(* PLC project OOP_Curso, Beckhoff Automation GmbH TwinCAT PLC Control 3.5.13.21 *)
(* stored: creationDateTime 2023-06-14T13:02:06.5620853, modificationDateTime 2023-06-14T13:02:06.5620853 *)

(* global variable list GVL_Exc *)
{attribute 'qualified_only'}
VAR_GLOBAL CONSTANT
    cMaxExc            : UINT := 10;
END_VAR
VAR_GLOBAL
    nExcIndex          : UINT;
    aExceptionHistory  : ARRAY[0..cMaxExc] OF __SYSTEM.ExceptionCode;
END_VAR

(* global variable list GVL *)
{attribute 'qualified_only'}
VAR_GLOBAL
    bGlobalTestFlag : BOOL;
END_VAR

INTERFACE I_Base EXTENDS __SYSTEM.IQueryInterface
METHOD Base : BOOL
VAR_INPUT
END_VAR
END_METHOD
END_INTERFACE

INTERFACE I_Derived EXTENDS I_Base
METHOD Derived : BOOL
VAR_INPUT
END_VAR
END_METHOD
END_INTERFACE

FUNCTION_BLOCK FB_Variante IMPLEMENTS I_Derived
VAR_INPUT
END_VAR
VAR_OUTPUT
END_VAR
VAR
END_VAR

            
          

{warning 'add method implementation '}
METHOD Base : BOOL
                  
                
END_METHOD

{warning 'add method implementation '}
METHOD Derived : BOOL
                  
                
END_METHOD
END_FUNCTION_BLOCK

PROGRAM QUERYPOINTER
//__QUERYPOINTER
VAR
    iDerived   : I_Derived;
    fbVariante : FB_Variante;
    bResult    : BOOL;
    bTest      : BOOL;
    pFB        : POINTER TO FB_Variante;
END_VAR

            //__QUERYPOINTER
iDerived := fbVariante;
bResult  := __QUERYPOINTER(iDerived, pFB);

IF bResult THEN
    bTest := pFB^.Derived();
END_IF
          
END_PROGRAM

FUNCTION F_SaveExceptionCode : BOOL
VAR_INPUT
    excInput           : __SYSTEM.ExceptionCode;
END_VAR

            // Log the thrown exception into the global exception history array
IF GVL_Exc.nExcIndex <= GVL_Exc.cMaxExc THEN
    GVL_Exc.aExceptionHistory[GVL_Exc.nExcIndex] := excInput;
    GVL_Exc.nExcIndex := GVL_Exc.nExcIndex + 1;
END_IF
          
END_FUNCTION

PROGRAM TRY_CATCH
//__TRY, __CATCH, __FINALLY, __ENDTRY
VAR
    nCounter1          : INT;
    nCounter2          : INT;
    nCounter_TRY1      : INT;
    nCounter_TRY2      : INT;
    nCounter_CATCH     : INT;    
    nCounter_FINALLY   : INT;
 
    exc                : __SYSTEM.ExceptionCode;
    lastExc            : __SYSTEM.ExceptionCode;
 
    pSample            : POINTER TO BOOL;
    bVar               : BOOL;
    nSample            : INT := 100;
    nDivisor           : INT;
END_VAR

            // -- !!! Available from TC3.1 build 4024 for 32-bit runtime systems !!!
////__TRY, __CATCH, __FINALLY, __ENDTRY 
//// Counter 1
//nCounter1 := nCounter1 + 1;
 
//// TRY-CATCH block
//__TRY
//    nCounter_TRY1 := nCounter_TRY1 + 1;
//    pSample^      := TRUE;                // 1. cycle: null pointer access leads to "access violation" exception
//    nSample       := nSample/nDivisor;    // 2. cycle: division by zero leads to "divide by zero" exception
//    nCounter_TRY2 := nCounter_TRY2 + 1;
 
//__CATCH(exc)
//    nCounter_CATCH    := nCounter_CATCH + 1;
 
//    // Exception logging
//    lastExc := exc;
//    F_SaveExceptionCode(excInput := exc);
 
//    // Correct the faulty variable values
//    IF (exc = __SYSTEM.ExceptionCode.RTSEXCPT_ACCESS_VIOLATION) AND (pSample = 0) THEN
//        pSample  := ADR(bVar);
// ELSIF ((exc = __SYSTEM.ExceptionCode.RTSEXCPT_DIVIDEBYZERO) OR (exc = __SYSTEM.ExceptionCode.RTSEXCPT_FPU_DIVIDEBYZERO)) AND (nDivisor = 0) THEN
//        nDivisor := 1;
//    END_IF
 
//__FINALLY
//    nCounter_FINALLY := nCounter_FINALLY + 1;
 
//__ENDTRY
 
//// Counter 2
//nCounter2 := nCounter2 + 1;
          
END_PROGRAM

PROGRAM VARINFO

VAR
    MyVarInfo : __SYSTEM.VAR_INFO;
    nVar      : INT;
END_VAR

            MyVarInfo := __VARINFO(nVar);
          
END_PROGRAM

PROGRAM TestAndSet1
VAR
    nLocalBlockedCounter : DINT;
END_VAR

            IF TestAndSet(GVL.bGlobalTestFlag) THEN
    (* bGlobalTestFlag was FALSE, nobody was blocking, NOW
    bGlobalTestFlag is set to TRUE and blocking others *)
    
    (* ... *)
    
    (* remove blocking by resetting the flag *) 
    GVL.bGlobalTestFlag := FALSE;
ELSE
    (* bGlobalTestFlag was TRUE, somebody is blocking *)
    nLocalBlockedCounter := nLocalBlockedCounter + 1;
    
    (* ... *)
END_IF



          
END_PROGRAM

PROGRAM _18_Otros_Operadores2

            
QUERYPOINTER();
TRY_CATCH();
VARINFO();
TestAndSet1();
          
END_PROGRAM
